Yaskawa INFORM job: blower_cylinder_program2.JBI

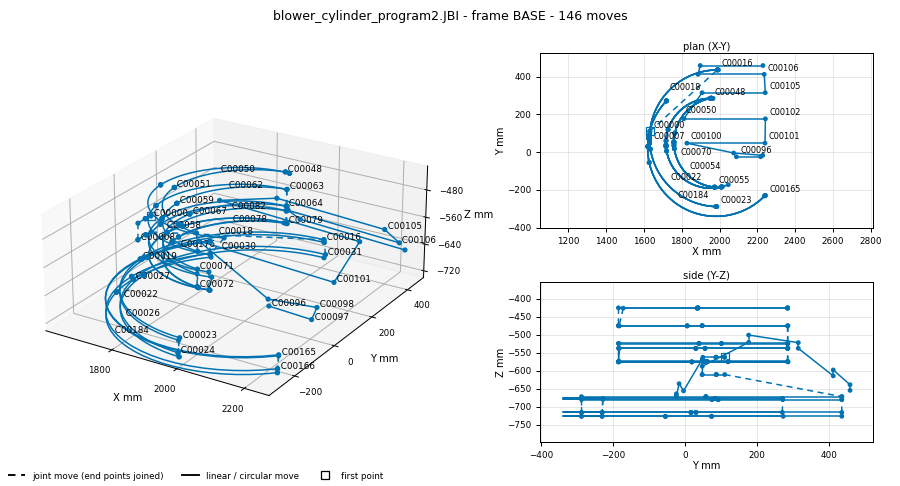
[picture p0: tool path of blower_cylinder_program2.JBI in frame BASE, 146 of 201 moves have a stored position in this frame; points joined in program order, loops and branches not executed]
/JOB
//NAME blower_cylinder_program2
//POS
///NPOS 190,0,190,0,0,0
///TOOL 0
///POSTYPE BASE
///RECTAN
///RCONF 0,0,0,0,0,0,0,0,0,0,0,0,0,0,0,0,0,0,0,0,0,0,0,0
C00000=1631.040523,109.687565,-562.117000,174.285929,-90.000000,5.000000
C00001=1631.040523,109.687565,-562.117000,174.285929,-90.000000,5.000000
C00002=1630.008214,97.187943,-562.117000,175.000000,-90.000000,5.000000
C00003=1629.444530,85.752258,-562.117000,175.000000,-90.000000,5.000000
C00004=1629.444530,85.752258,-562.117000,175.000000,-90.000000,5.000000
C00005=1629.444530,85.752258,-562.117000,175.000000,-90.000000,5.000000
C00006=1629.333691,65.522471,-562.117000,-175.000000,-90.000000,5.000000
C00007=1630.058515,49.363077,-562.117000,-175.000000,-89.999999,5.000000
C00008=1630.198827,47.360412,-610.141500,-175.000000,-89.999999,5.000000
C00009=1630.198827,47.360412,-610.141500,-175.000000,-89.999999,5.000000
C00010=1629.243181,72.855179,-610.141500,-175.000000,-90.000000,5.000000
C00011=1629.466653,86.396553,-610.141500,175.000000,-90.000000,5.000000
C00012=1629.466653,86.396553,-610.141500,175.000000,-90.000000,5.000000
C00013=1629.466653,86.396553,-610.141500,175.000000,-90.000000,5.000000
C00014=1630.172126,99.581103,-610.141500,175.000000,-90.000000,5.000000
C00015=1631.080525,110.085124,-610.141500,174.222670,-90.000000,5.000000
C00016=1988.362900,435.544640,-671.548000,90.440036,-90.000000,5.000000
C00017=1988.362900,435.544640,-671.548000,90.440036,-90.000000,5.000000
C00018=1715.116522,307.709542,-671.548000,139.703942,-89.999999,5.000000
C00019=1629.590499,57.783708,-671.548000,-175.000000,-90.000000,5.000000
C00020=1629.590499,57.783708,-671.548000,-175.000000,-90.000000,5.000000
C00021=1629.590499,57.783708,-671.548000,-175.000000,-90.000000,5.000000
C00022=1722.107790,-168.402623,-671.548000,-138.021392,-90.000000,5.000000
C00023=1986.333631,-288.212739,-671.548000,-90.761327,-90.000000,5.000000
C00024=1980.447685,-288.086633,-715.494500,-91.693411,-90.000000,5.000000
C00025=1980.447685,-288.086633,-715.494500,-91.693411,-90.000000,5.000000
C00026=1739.500917,-186.437414,-715.494500,-134.053840,-90.000000,5.000000
C00027=1633.810488,16.335257,-715.494500,-170.886748,-89.999999,5.000000
C00028=1633.810488,16.335257,-715.494500,-170.886748,-89.999999,5.000000
C00029=1633.810488,16.335257,-715.494500,-170.886748,-89.999999,5.000000
C00030=1719.796907,313.119903,-715.494500,138.571326,-90.000000,5.000000
C00031=1994.191551,435.542467,-715.494500,89.517238,-89.999999,5.000000
C00032=1989.404478,435.551141,-679.645460,-175.000000,-60.000000,-89.724869
C00033=1989.404478,435.551141,-679.645460,-175.000000,-60.000000,-89.724869
C00034=1742.952661,337.043838,-679.645460,175.000000,-60.000000,-46.701746
C00035=1629.697411,91.799312,-679.645460,175.000000,-60.000000,-5.000000
C00036=1629.697411,91.799312,-679.645460,175.000000,-60.000000,-5.000000
C00037=1629.697411,91.799312,-679.645460,175.000000,-60.000000,-5.000000
C00038=1718.918651,-164.810402,-679.645460,175.000000,-60.000000,41.218098
C00039=1982.731197,-288.146931,-679.645460,-175.000000,-60.000000,88.668240
C00040=1983.607859,-288.166248,-726.148460,175.000000,-60.000000,88.807067
C00041=1983.607859,-288.166248,-726.148460,175.000000,-60.000000,88.807067
C00042=1731.491014,-178.441537,-726.148460,-175.000000,-60.000000,44.154260
C00043=1629.242368,73.427735,-726.148460,175.000000,-60.000000,5.000000
C00044=1629.242368,73.427735,-726.148460,175.000000,-60.000000,5.000000
C00045=1629.242368,73.427735,-726.148460,175.000000,-60.000000,5.000000
C00046=1733.297996,327.600045,-726.148460,-175.000000,-60.000000,-44.563444
C00047=1989.524610,435.551697,-726.148460,175.000000,-60.000000,-89.743888
C00048=1951.500120,284.949500,-424.583000,100.823768,-89.999999,5.000000
C00049=1951.500120,284.949500,-424.583000,100.823768,-89.999999,5.000000
C00050=1799.733446,185.412825,-424.583000,145.694229,-90.000000,5.000000
C00051=1758.900904,35.496503,-424.583000,-175.000000,-90.000000,5.000000
C00052=1758.900904,35.496503,-424.583000,-175.000000,-90.000000,5.000000
C00053=1758.900904,35.496503,-424.583000,-175.000000,-90.000000,5.000000
C00054=1821.806950,-110.298412,-424.583000,-137.156322,-89.999999,5.000000
C00055=1972.212153,-185.181050,-424.583000,-95.778594,-90.000000,5.000000
C00056=1975.163697,-185.461165,-474.319000,-95.064200,-89.999999,5.000000
C00057=1975.163697,-185.461165,-474.319000,-95.064200,-89.999999,5.000000
C00058=1821.392397,-109.850266,-474.319000,-137.303422,-89.999999,5.000000
C00059=1758.402792,47.374762,-474.319000,-175.000000,-90.000000,5.000000
C00060=1758.402792,47.374762,-474.319000,-175.000000,-90.000000,5.000000
C00061=1758.402792,47.374762,-474.319000,-175.000000,-90.000000,5.000000
C00062=1813.745711,203.936859,-474.319000,140.095354,-90.000000,5.000000
C00063=1956.985939,285.931842,-474.319000,99.480867,-90.000000,5.000000
C00064=1954.568672,285.515334,-523.825000,100.071909,-90.000000,5.000000
C00065=1954.568672,285.515334,-523.825000,100.071909,-90.000000,5.000000
C00066=1800.113961,185.968824,-523.825000,145.531886,-90.000000,5.000000
C00067=1763.606613,101.028958,-523.825000,167.951827,-90.000000,5.000000
C00068=1763.606613,101.028958,-523.825000,167.951827,-90.000000,5.000000
C00069=1763.606613,101.028958,-523.825000,167.951827,-90.000000,5.000000
C00070=1774.472432,-34.622591,-523.825000,-158.792489,-90.000000,5.000000
C00071=1974.161805,-185.370243,-523.825000,-95.306604,-90.000000,5.000000
C00072=1972.366476,-185.196616,-573.993000,-95.741220,-90.000000,5.000000
C00073=1972.366476,-185.196616,-573.993000,-95.741220,-90.000000,5.000000
C00074=1805.880129,-91.214728,-573.993000,-143.148416,-90.000000,5.000000
C00075=1758.377712,53.453915,-573.993000,175.000000,-90.000000,5.000000
C00076=1758.377712,53.453915,-573.993000,175.000000,-90.000000,5.000000
C00077=1758.377712,53.453915,-573.993000,175.000000,-90.000000,5.000000
C00078=1821.730072,213.005923,-573.993000,137.183571,-90.000000,5.000000
C00079=1954.737393,285.545239,-573.993000,100.030621,-90.000000,5.000000
C00080=1954.939494,285.580897,-537.232460,175.000000,-60.000000,-80.018829
C00081=1954.939494,285.580897,-537.232460,175.000000,-60.000000,-80.018829
C00082=1819.578522,210.652337,-537.232460,175.000000,-60.000000,-42.048057
C00083=1758.400787,55.295319,-537.232460,-175.000000,-60.000000,-5.000000
C00084=1758.400787,55.295319,-537.232460,-175.000000,-60.000000,-5.000000
C00085=1758.400787,55.295319,-537.232460,-175.000000,-60.000000,-5.000000
C00086=1801.050561,-84.532692,-537.232460,175.000000,-60.000000,34.864881
C00087=1972.684728,-185.228397,-537.232460,-175.000000,-60.000000,84.335846
C00088=1976.970675,-185.614353,-575.051960,175.000000,-60.000000,85.372767
C00089=1976.970675,-185.614353,-575.051960,175.000000,-60.000000,85.372767
C00090=1824.259860,-112.903672,-575.051960,-175.000000,-60.000000,43.705898
C00091=1760.661540,18.454371,-575.051960,-175.000000,-60.000000,7.962927
C00092=1760.661540,18.454371,-575.051960,-175.000000,-60.000000,7.962927
C00093=1760.661540,18.454371,-575.051960,-175.000000,-60.000000,7.962927
C00094=1790.604013,170.940048,-575.051960,-175.000000,-60.000000,-30.181721
C00095=1957.730202,286.054921,-575.051960,-175.000000,-60.000000,-80.700904
C00096=2089.306045,-24.353058,-663.745553,175.000000,-60.000000,90.065286
C00097=2217.470262,-24.353051,-669.800856,175.000000,-60.000000,90.065286
C00098=2228.297277,-16.748565,-635.673601,-175.000000,-60.000000,91.170202
C00099=2074.711330,-4.438705,-655.515790,175.000000,-66.623448,91.170202
C00100=1827.048359,47.582539,-567.652515,175.000000,-44.740427,92.732701
C00101=2240.740165,47.582562,-587.197981,175.000000,-44.740427,92.732701
C00102=2242.656280,176.551574,-520.760389,-170.133186,5.000000,5.000000
C00103=1810.757184,176.551550,-500.354693,-170.133186,5.000000,5.000000
C00104=1907.631611,314.643219,-521.482904,156.457092,5.000000,-5.000000
C00105=2242.006831,314.643237,-537.280944,156.457092,5.000000,-5.000000
C00106=2236.445037,411.851577,-613.890742,175.000000,-53.159924,-92.028486
C00107=1886.225138,411.851557,-597.344097,175.000000,-53.159924,-92.028486
C00108=1897.676258,458.517871,-638.458617,175.000000,-60.000000,-90.549119
C00109=2229.933616,458.517890,-654.156596,175.000000,-60.000000,-90.549119
C00110=1964.745052,284.514995,-425.665500,87.414352,-90.000000,5.000000
C00111=1964.745052,284.514995,-425.665500,87.414352,-90.000000,5.000000
C00112=1791.215190,220.283714,-425.665500,133.209250,-89.999999,5.000000
C00113=1716.607937,33.630447,-425.665500,-175.000000,-89.999999,5.000000
C00114=1716.607937,33.630447,-425.665500,-175.000000,-89.999999,5.000000
C00115=1716.607937,33.630447,-425.665500,-175.000000,-89.999999,5.000000
C00116=1823.917544,-152.063706,-425.665500,-123.170715,-89.999999,5.000000
C00117=2046.235000,-172.202170,-425.665500,-67.181224,-90.000000,5.000000
C00118=2011.577078,-183.740457,-474.764500,-75.991595,-89.999999,5.000000
C00119=2011.577078,-183.740457,-474.764500,-75.991595,-89.999999,5.000000
C00120=1824.819666,-152.650471,-474.764500,-122.911408,-89.999999,5.000000
C00121=1719.835816,5.738371,-474.764500,-170.013885,-90.000000,5.000000
C00122=1719.835816,5.738371,-474.764500,-170.013885,-90.000000,5.000000
C00123=1719.835816,5.738371,-474.764500,-170.013885,-90.000000,5.000000
C00124=1790.195887,219.320542,-474.764500,133.547165,-89.999999,5.000000
C00125=1955.860288,284.749946,-474.764500,89.556068,-90.000000,5.000000
C00126=1957.611787,284.729923,-523.805000,89.134004,-90.000000,5.000000
C00127=1957.611787,284.729923,-523.805000,89.134004,-90.000000,5.000000
C00128=1776.978575,205.713095,-523.805000,138.119319,-89.999999,5.000000
C00129=1716.378968,38.651546,-523.805000,-175.000000,-90.000000,5.000000
C00130=1716.378968,38.651546,-523.805000,-175.000000,-90.000000,5.000000
C00131=1716.378968,38.651546,-523.805000,-175.000000,-90.000000,5.000000
C00132=1814.172099,-145.341475,-523.805000,-126.023698,-89.999999,5.000000
C00133=2008.136089,-184.571770,-523.805000,-76.844586,-90.000000,5.000000
C00134=2008.342338,-184.523467,-573.820000,-76.793544,-90.000000,5.000000
C00135=2008.342338,-184.523467,-573.820000,-76.793544,-90.000000,5.000000
C00136=1814.343644,-145.466101,-573.820000,-125.972606,-89.999999,5.000000
C00137=1716.639179,60.859270,-573.820000,175.000000,-90.000000,5.000000
C00138=1716.639179,60.859270,-573.820000,175.000000,-90.000000,5.000000
C00139=1716.639179,60.859270,-573.820000,175.000000,-90.000000,5.000000
C00140=1783.695738,212.899774,-573.820000,135.748834,-90.000000,5.000000
C00141=1957.832909,284.726478,-573.820000,89.080717,-89.999999,5.000000
C00142=1956.063429,284.748285,-537.333960,175.000000,-60.000000,-90.492882
C00143=1956.063429,284.748285,-537.333960,175.000000,-60.000000,-90.492882
C00144=1793.267213,222.188698,-537.333960,175.000000,-60.000000,-47.465422
C00145=1716.866308,29.634015,-537.333960,-175.000000,-60.000000,5.000000
C00146=1716.866308,29.634015,-537.333960,-175.000000,-60.000000,5.000000
C00147=1716.866308,29.634015,-537.333960,-175.000000,-60.000000,5.000000
C00148=1807.150688,-140.034277,-537.333960,-175.000000,-60.000000,51.855399
C00149=2015.398585,-182.753292,-537.333960,-175.000000,-60.000000,104.959459
C00150=2010.433958,-184.022643,-574.408960,175.000000,-60.000000,103.724694
C00151=2010.433958,-184.022643,-574.408960,175.000000,-60.000000,103.724694
C00152=1758.658341,-88.586161,-574.408960,175.000000,-60.000000,34.756508
C00153=1727.512341,119.337756,-574.408960,175.000000,-60.000000,-17.717932
C00154=1727.512341,119.337756,-574.408960,175.000000,-60.000000,-17.717932
C00155=1727.512341,119.337756,-574.408960,175.000000,-60.000000,-17.717932
C00156=1818.979093,242.691740,-574.408960,-175.000000,-60.000000,-55.395801
C00157=1948.601509,284.695386,-574.408960,175.000000,-60.000000,-88.694764
C00158=1718.289686,270.799606,-676.690500,136.574254,-90.000000,5.000000
C00159=1718.289686,270.799606,-676.690500,136.574254,-90.000000,5.000000
C00160=1655.911050,180.792580,-676.690500,153.978586,-90.000000,5.000000
C00161=1624.512379,83.659193,-676.690500,170.194237,-90.000000,5.000000
C00162=1624.512379,83.659193,-676.690500,170.194237,-90.000000,5.000000
C00163=1624.512379,83.659193,-676.690500,170.194237,-90.000000,5.000000
C00164=1644.313839,-110.375076,-676.690500,-158.540358,-90.000000,5.000000
C00165=2242.018060,-228.787332,-676.690500,-43.871381,-90.000000,5.000000
C00166=2240.253119,-230.610376,-715.292500,-44.273105,-89.999999,5.000000
C00167=2240.253119,-230.610376,-715.292500,-44.273105,-89.999999,5.000000
C00168=1639.607599,-97.713833,-715.292500,-160.679000,-90.000000,5.000000
C00169=1619.314173,30.044393,-715.292500,175.000000,-90.000000,5.000000
C00170=1619.314173,30.044393,-715.292500,175.000000,-90.000000,5.000000
C00171=1619.314173,30.044393,-715.292500,175.000000,-90.000000,5.000000
C00172=1643.442938,152.186837,-715.292500,158.920449,-90.000000,5.000000
C00173=1717.643970,270.115616,-715.292500,136.723175,-89.999999,5.000000
C00174=1718.984125,271.531248,-679.384960,-175.000000,-60.000000,-43.585448
C00175=1718.984125,271.531248,-679.384960,-175.000000,-60.000000,-43.585448
C00176=1662.611066,193.839210,-679.384960,175.000000,-60.000000,-28.343556
C00177=1623.069692,74.634311,-679.384960,175.000000,-60.000000,-8.358770
C00178=1623.069692,74.634311,-679.384960,175.000000,-60.000000,-8.358770
C00179=1623.069692,74.634311,-679.384960,175.000000,-60.000000,-8.358770
C00180=1633.197058,-77.562383,-679.384960,-175.000000,-60.000000,15.972617
C00181=2241.912484,-228.897104,-679.384960,175.000000,-60.000000,136.104507
C00182=2240.003412,-230.866247,-726.338960,175.000000,-60.000000,135.670292
C00183=2240.003412,-230.866247,-726.338960,175.000000,-60.000000,135.670292
C00184=1759.939773,-264.416714,-726.338960,175.000000,-60.000000,52.325229
C00185=1627.509593,-54.966023,-726.338960,175.000000,-60.000000,12.282959
C00186=1627.509593,-54.966023,-726.338960,175.000000,-60.000000,12.282959
C00187=1627.509593,-54.966023,-726.338960,175.000000,-60.000000,12.282959
C00188=1632.511691,119.184999,-726.338960,175.000000,-60.000000,-15.573440
C00189=1720.027963,272.623370,-726.338960,-175.000000,-60.000000,-43.824627
///POSTYPE PULSE
///PULSE
EX00000=91136.0
EX00001=94208.0
EX00002=113664.0
EX00003=282624.0
EX00004=323584.0
///POSTYPE PULSE
///PULSE
EC00000=91136.0
EC00001=91136.0
EC00002=91136.0
EC00003=91136.0
EC00004=91136.0
EC00005=91136.0
EC00006=91136.0
EC00007=91136.0
EC00008=91136.0
EC00009=91136.0
EC00010=91136.0
EC00011=91136.0
EC00012=91136.0
EC00013=91136.0
EC00014=91136.0
EC00015=91136.0
EC00016=91136.0
EC00017=91136.0
EC00018=91136.0
EC00019=91136.0
EC00020=91136.0
EC00021=91136.0
EC00022=91136.0
EC00023=91136.0
EC00024=91136.0
EC00025=91136.0
EC00026=91136.0
EC00027=91136.0
EC00028=91136.0
EC00029=91136.0
EC00030=91136.0
EC00031=91136.0
EC00032=91136.0
EC00033=91136.0
EC00034=91136.0
EC00035=91136.0
EC00036=91136.0
EC00037=91136.0
EC00038=91136.0
EC00039=91136.0
EC00040=91136.0
EC00041=91136.0
EC00042=91136.0
EC00043=91136.0
EC00044=91136.0
EC00045=91136.0
EC00046=91136.0
EC00047=91136.0
EC00048=94208.0
EC00049=94208.0
EC00050=94208.0
EC00051=94208.0
EC00052=94208.0
EC00053=94208.0
EC00054=94208.0
EC00055=94208.0
EC00056=94208.0
EC00057=94208.0
EC00058=94208.0
EC00059=94208.0
EC00060=94208.0
EC00061=94208.0
EC00062=94208.0
EC00063=94208.0
EC00064=94208.0
EC00065=94208.0
EC00066=94208.0
EC00067=94208.0
EC00068=94208.0
EC00069=94208.0
EC00070=94208.0
EC00071=94208.0
EC00072=94208.0
EC00073=94208.0
EC00074=94208.0
EC00075=94208.0
EC00076=94208.0
EC00077=94208.0
EC00078=94208.0
EC00079=94208.0
EC00080=94208.0
EC00081=94208.0
EC00082=94208.0
EC00083=94208.0
EC00084=94208.0
EC00085=94208.0
EC00086=94208.0
EC00087=94208.0
EC00088=94208.0
EC00089=94208.0
EC00090=94208.0
EC00091=94208.0
EC00092=94208.0
EC00093=94208.0
EC00094=94208.0
EC00095=94208.0
EC00096=113664.0
EC00097=113664.0
EC00098=113664.0
EC00099=113664.0
EC00100=113664.0
EC00101=113664.0
EC00102=113664.0
EC00103=113664.0
EC00104=113664.0
EC00105=113664.0
EC00106=113664.0
EC00107=113664.0
EC00108=113664.0
EC00109=113664.0
EC00110=282624.0
EC00111=282624.0
EC00112=282624.0
EC00113=282624.0
EC00114=282624.0
EC00115=282624.0
EC00116=282624.0
EC00117=282624.0
EC00118=282624.0
EC00119=282624.0
EC00120=282624.0
EC00121=282624.0
EC00122=282624.0
EC00123=282624.0
EC00124=282624.0
EC00125=282624.0
EC00126=282624.0
EC00127=282624.0
EC00128=282624.0
EC00129=282624.0
EC00130=282624.0
EC00131=282624.0
EC00132=282624.0
EC00133=282624.0
EC00134=282624.0
EC00135=282624.0
EC00136=282624.0
EC00137=282624.0
EC00138=282624.0
EC00139=282624.0
EC00140=282624.0
EC00141=282624.0
EC00142=282624.0
EC00143=282624.0
EC00144=282624.0
EC00145=282624.0
EC00146=282624.0
EC00147=282624.0
EC00148=282624.0
EC00149=282624.0
EC00150=282624.0
EC00151=282624.0
EC00152=282624.0
EC00153=282624.0
EC00154=282624.0
EC00155=282624.0
EC00156=282624.0
EC00157=282624.0
EC00158=323584.0
EC00159=323584.0
EC00160=323584.0
EC00161=323584.0
EC00162=323584.0
EC00163=323584.0
EC00164=323584.0
EC00165=323584.0
EC00166=323584.0
EC00167=323584.0
EC00168=323584.0
EC00169=323584.0
EC00170=323584.0
EC00171=323584.0
EC00172=323584.0
EC00173=323584.0
EC00174=323584.0
EC00175=323584.0
EC00176=323584.0
EC00177=323584.0
EC00178=323584.0
EC00179=323584.0
EC00180=323584.0
EC00181=323584.0
EC00182=323584.0
EC00183=323584.0
EC00184=323584.0
EC00185=323584.0
EC00186=323584.0
EC00187=323584.0
EC00188=323584.0
EC00189=323584.0
//INST
///DATE 2023/08/15 16:42
///ATTR SC,RW,RJ
////FRAME BASE
///GROUP1 RB1,ST1
NOP
MOVJ P009 EX000 VJ=15.00
MOVJ C00000 EC00000 VJ=15.0
CALL JOB:SPYON
MOVC C00001 EC00001 V=150.0
MOVC C00002 EC00002 V=150.0
MOVC C00003 EC00003 V=150.0
MOVJ C00004 EC00004 VJ=15.0
MOVC C00005 EC00005 V=150.0
MOVC C00006 EC00006 V=150.0
MOVC C00007 EC00007 V=150.0
MOVJ C00008 EC00008 VJ=15.0
MOVC C00009 EC00009 V=150.0
MOVC C00010 EC00010 V=150.0
MOVC C00011 EC00011 V=150.0
MOVJ C00012 EC00012 VJ=15.0
MOVC C00013 EC00013 V=150.0
MOVC C00014 EC00014 V=150.0
MOVC C00015 EC00015 V=150.0
MOVJ C00016 EC00016 VJ=15.0
MOVC C00017 EC00017 V=150.0
MOVC C00018 EC00018 V=150.0
MOVC C00019 EC00019 V=150.0
MOVJ C00020 EC00020 VJ=15.0
MOVC C00021 EC00021 V=150.0
MOVC C00022 EC00022 V=150.0
MOVC C00023 EC00023 V=150.0
MOVJ C00024 EC00024 VJ=15.0
MOVC C00025 EC00025 V=150.0
MOVC C00026 EC00026 V=150.0
MOVC C00027 EC00027 V=150.0
MOVJ C00028 EC00028 VJ=15.0
MOVC C00029 EC00029 V=150.0
MOVC C00030 EC00030 V=150.0
MOVC C00031 EC00031 V=150.0
MOVJ C00032 EC00032 VJ=15.0
MOVC C00033 EC00033 V=150.0
MOVC C00034 EC00034 V=150.0
MOVC C00035 EC00035 V=150.0
MOVJ C00036 EC00036 VJ=15.0
MOVC C00037 EC00037 V=150.0
MOVC C00038 EC00038 V=150.0
MOVC C00039 EC00039 V=150.0
MOVJ C00040 EC00040 VJ=15.0
MOVC C00041 EC00041 V=150.0
MOVC C00042 EC00042 V=150.0
MOVC C00043 EC00043 V=150.0
MOVJ C00044 EC00044 VJ=15.0
MOVC C00045 EC00045 V=150.0
MOVC C00046 EC00046 V=150.0
MOVC C00047 EC00047 V=150.0
CALL JOB:SPYOF
MOVJ P009 VJ=15.00
MOVL P009 EX00000 V=150.0
MOVJ C00048 EC00048 VJ=15.0
CALL JOB:SPYON
MOVC C00049 EC00049 V=150.0
MOVC C00050 EC00050 V=150.0
MOVC C00051 EC00051 V=150.0
MOVJ C00052 EC00052 VJ=15.0
MOVC C00053 EC00053 V=150.0
MOVC C00054 EC00054 V=150.0
MOVC C00055 EC00055 V=150.0
MOVJ C00056 EC00056 VJ=15.0
MOVC C00057 EC00057 V=150.0
MOVC C00058 EC00058 V=150.0
MOVC C00059 EC00059 V=150.0
MOVJ C00060 EC00060 VJ=15.0
MOVC C00061 EC00061 V=150.0
MOVC C00062 EC00062 V=150.0
MOVC C00063 EC00063 V=150.0
MOVJ C00064 EC00064 VJ=15.0
MOVC C00065 EC00065 V=150.0
MOVC C00066 EC00066 V=150.0
MOVC C00067 EC00067 V=150.0
MOVJ C00068 EC00068 VJ=15.0
MOVC C00069 EC00069 V=150.0
MOVC C00070 EC00070 V=150.0
MOVC C00071 EC00071 V=150.0
MOVJ C00072 EC00072 VJ=15.0
MOVC C00073 EC00073 V=150.0
MOVC C00074 EC00074 V=150.0
MOVC C00075 EC00075 V=150.0
MOVJ C00076 EC00076 VJ=15.0
MOVC C00077 EC00077 V=150.0
MOVC C00078 EC00078 V=150.0
MOVC C00079 EC00079 V=150.0
MOVJ C00080 EC00080 VJ=15.0
MOVC C00081 EC00081 V=150.0
MOVC C00082 EC00082 V=150.0
MOVC C00083 EC00083 V=150.0
MOVJ C00084 EC00084 VJ=15.0
MOVC C00085 EC00085 V=150.0
MOVC C00086 EC00086 V=150.0
MOVC C00087 EC00087 V=150.0
MOVJ C00088 EC00088 VJ=15.0
MOVC C00089 EC00089 V=150.0
MOVC C00090 EC00090 V=150.0
MOVC C00091 EC00091 V=150.0
MOVJ C00092 EC00092 VJ=15.0
MOVC C00093 EC00093 V=150.0
MOVC C00094 EC00094 V=150.0
MOVC C00095 EC00095 V=150.0
CALL JOB:SPYOF
MOVJ P009 VJ=15.00
MOVL P009 EX00001 V=150.0
MOVJ C00096 EC00096 VJ=15.0
CALL JOB:SPYON
MOVL C00097 EC00097 V=150.0
MOVL C00098 EC00098 V=150.0
MOVL C00099 EC00099 V=150.0
MOVL C00100 EC00100 V=150.0
MOVL C00101 EC00101 V=150.0
MOVL C00102 EC00102 V=150.0
MOVL C00103 EC00103 V=150.0
MOVL C00104 EC00104 V=150.0
MOVL C00105 EC00105 V=150.0
MOVL C00106 EC00106 V=150.0
MOVL C00107 EC00107 V=150.0
MOVL C00108 EC00108 V=150.0
MOVL C00109 EC00109 V=150.0
CALL JOB:SPYOF
MOVJ P009 VJ=15.00
MOVL P009 EX00002 V=150.0
MOVJ C00110 EC00110 VJ=15.0
CALL JOB:SPYON
MOVC C00111 EC00111 V=150.0
MOVC C00112 EC00112 V=150.0
MOVC C00113 EC00113 V=150.0
MOVJ C00114 EC00114 VJ=15.0
MOVC C00115 EC00115 V=150.0
MOVC C00116 EC00116 V=150.0
MOVC C00117 EC00117 V=150.0
MOVJ C00118 EC00118 VJ=15.0
MOVC C00119 EC00119 V=150.0
MOVC C00120 EC00120 V=150.0
MOVC C00121 EC00121 V=150.0
MOVJ C00122 EC00122 VJ=15.0
MOVC C00123 EC00123 V=150.0
MOVC C00124 EC00124 V=150.0
MOVC C00125 EC00125 V=150.0
MOVJ C00126 EC00126 VJ=15.0
MOVC C00127 EC00127 V=150.0
MOVC C00128 EC00128 V=150.0
MOVC C00129 EC00129 V=150.0
MOVJ C00130 EC00130 VJ=15.0
MOVC C00131 EC00131 V=150.0
MOVC C00132 EC00132 V=150.0
MOVC C00133 EC00133 V=150.0
MOVJ C00134 EC00134 VJ=15.0
MOVC C00135 EC00135 V=150.0
MOVC C00136 EC00136 V=150.0
MOVC C00137 EC00137 V=150.0
MOVJ C00138 EC00138 VJ=15.0
MOVC C00139 EC00139 V=150.0
MOVC C00140 EC00140 V=150.0
MOVC C00141 EC00141 V=150.0
MOVJ C00142 EC00142 VJ=15.0
MOVC C00143 EC00143 V=150.0
MOVC C00144 EC00144 V=150.0
MOVC C00145 EC00145 V=150.0
MOVJ C00146 EC00146 VJ=15.0
MOVC C00147 EC00147 V=150.0
MOVC C00148 EC00148 V=150.0
MOVC C00149 EC00149 V=150.0
MOVJ C00150 EC00150 VJ=15.0
MOVC C00151 EC00151 V=150.0
MOVC C00152 EC00152 V=150.0
MOVC C00153 EC00153 V=150.0
MOVJ C00154 EC00154 VJ=15.0
MOVC C00155 EC00155 V=150.0
MOVC C00156 EC00156 V=150.0
MOVC C00157 EC00157 V=150.0
CALL JOB:SPYOF
MOVJ P009 VJ=15.00
MOVL P009 EX00003 V=150.0
MOVJ C00158 EC00158 VJ=15.0
CALL JOB:SPYON
MOVC C00159 EC00159 V=150.0
MOVC C00160 EC00160 V=150.0
MOVC C00161 EC00161 V=150.0
MOVJ C00162 EC00162 VJ=15.0
MOVC C00163 EC00163 V=150.0
MOVC C00164 EC00164 V=150.0
MOVC C00165 EC00165 V=150.0
MOVJ C00166 EC00166 VJ=15.0
MOVC C00167 EC00167 V=150.0
MOVC C00168 EC00168 V=150.0
MOVC C00169 EC00169 V=150.0
MOVJ C00170 EC00170 VJ=15.0
MOVC C00171 EC00171 V=150.0
MOVC C00172 EC00172 V=150.0
MOVC C00173 EC00173 V=150.0
MOVJ C00174 EC00174 VJ=15.0
MOVC C00175 EC00175 V=150.0
MOVC C00176 EC00176 V=150.0
MOVC C00177 EC00177 V=150.0
MOVJ C00178 EC00178 VJ=15.0
MOVC C00179 EC00179 V=150.0
MOVC C00180 EC00180 V=150.0
MOVC C00181 EC00181 V=150.0
MOVJ C00182 EC00182 VJ=15.0
MOVC C00183 EC00183 V=150.0
MOVC C00184 EC00184 V=150.0
MOVC C00185 EC00185 V=150.0
MOVJ C00186 EC00186 VJ=15.0
MOVC C00187 EC00187 V=150.0
MOVC C00188 EC00188 V=150.0
MOVC C00189 EC00189 V=150.0
CALL JOB:SPYOF
MOVJ P009 VJ=15.00
MOVL P009 EX00004 V=150.0
END
